{attribute addProperty BoxType "EK1122-0000-0018"}
{attribute addProperty Id "Beckhoff_EL37xxsub_EK1100EK1100_179A0949162"}
{attribute addProperty CRC "913456052"}
{attribute addProperty SizeInBites "16"}
{attribute addProperty SizeInBytes "2"}
TYPE Beckhoff_EL37xxEK1122_36723BB4 EXTENDS EK1122_179A0949 :
STRUCT
	{attribute addProperty Name "Beckhoff_EL37xxsub_EK1100"}
	Beckhoff_EL37xxsub_EK1100 : EK1100_179A0949;
END_STRUCT
END_TYPE

(* stored: Version 1.2.0.0, ProductVersion 3.1.4024.9
   DUT Beckhoff_EL37xxEK1122_36723BB4: Id {156a88e9-df59-4ad5-b230-6b727e34ddcc} *)
